FUNCTION_BLOCK FB_SineActivation_SC
VAR_INPUT
	bSineEnable			: BOOL;
	fStartPos_error		: LREAL;
END_VAR
VAR_OUTPUT
	bEnable				: BOOL;
END_VAR
VAR
	bStartPosOK			: BOOL;
END_VAR

IF ABS(fStartPos_error) < 0.2 THEN
	bStartPosOK := TRUE;
ELSIF NOT (G_IO.bStartButton) THEN
	bStartPosOK := FALSE;
END_IF

IF NOT(G_IO.bStartButton) THEN
	bEnable := FALSE;
	G_Engineer_HMI.bSecondarySineMotionEnable := FALSE;
	ELSIF bStartPosOK AND bSineEnable THEN
		bEnable := TRUE;
END_IF

END_FUNCTION_BLOCK

(* stored: Version 1.1.0.1
   POU FB_SineActivation_SC: Id {388698fb-0617-452b-a3fa-1efbe5cd9087}, SpecialFunc None *)
